KUKA KRL program: TestCutThreshold.src

&ACCESS RVEO
&REL 4
&PARAM EDITMASK = *
&PARAM TEMPLATE = C:\KRC\Roboter\Template\vorgabe
&PARAM DISKPATH = KRC:\R1\Program\LeafProfiles
DEF TestCutThreshold( )

   BAS(#INITMOV)
   ChangeStation(#HomePos)
   ChangeStation(#MillTable)

   ChangeStation(#CutRight)
   CutRight(#Leaf90,grShortProfileRefX,135)
   HALT
   ChangeStation(#CutRight)
   ChangeStation(#MillTable)

   ChangeStation(#HomePos)

END
